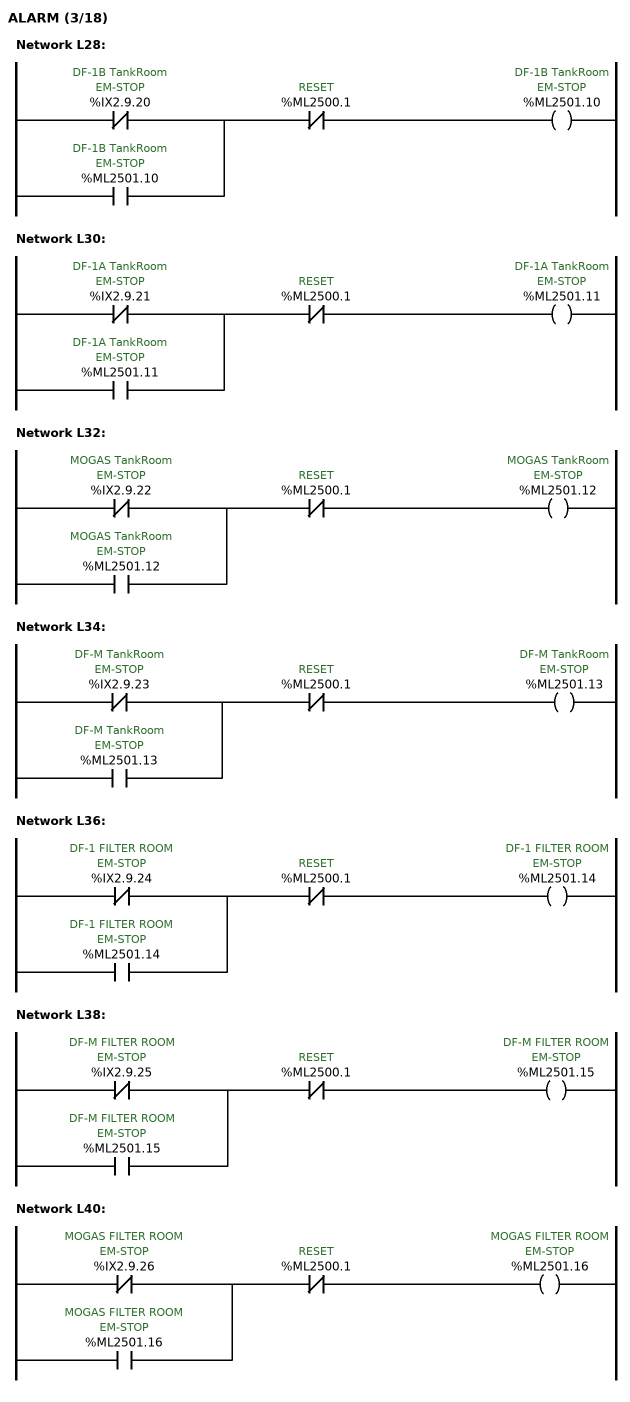
(* Rung L28 *)
%ML2501.10 := (NOT %IX2.9.20 OR %ML2501.10) AND NOT %ML2500.1;
(* Rung L30 *)
%ML2501.11 := (NOT %IX2.9.21 OR %ML2501.11) AND NOT %ML2500.1;
(* Rung L32 *)
%ML2501.12 := (NOT %IX2.9.22 OR %ML2501.12) AND NOT %ML2500.1;
(* Rung L34 *)
%ML2501.13 := (NOT %IX2.9.23 OR %ML2501.13) AND NOT %ML2500.1;
(* Rung L36 *)
%ML2501.14 := (NOT %IX2.9.24 OR %ML2501.14) AND NOT %ML2500.1;
(* Rung L38 *)
%ML2501.15 := (NOT %IX2.9.25 OR %ML2501.15) AND NOT %ML2500.1;
(* Rung L40 *)
%ML2501.16 := (NOT %IX2.9.26 OR %ML2501.16) AND NOT %ML2500.1;

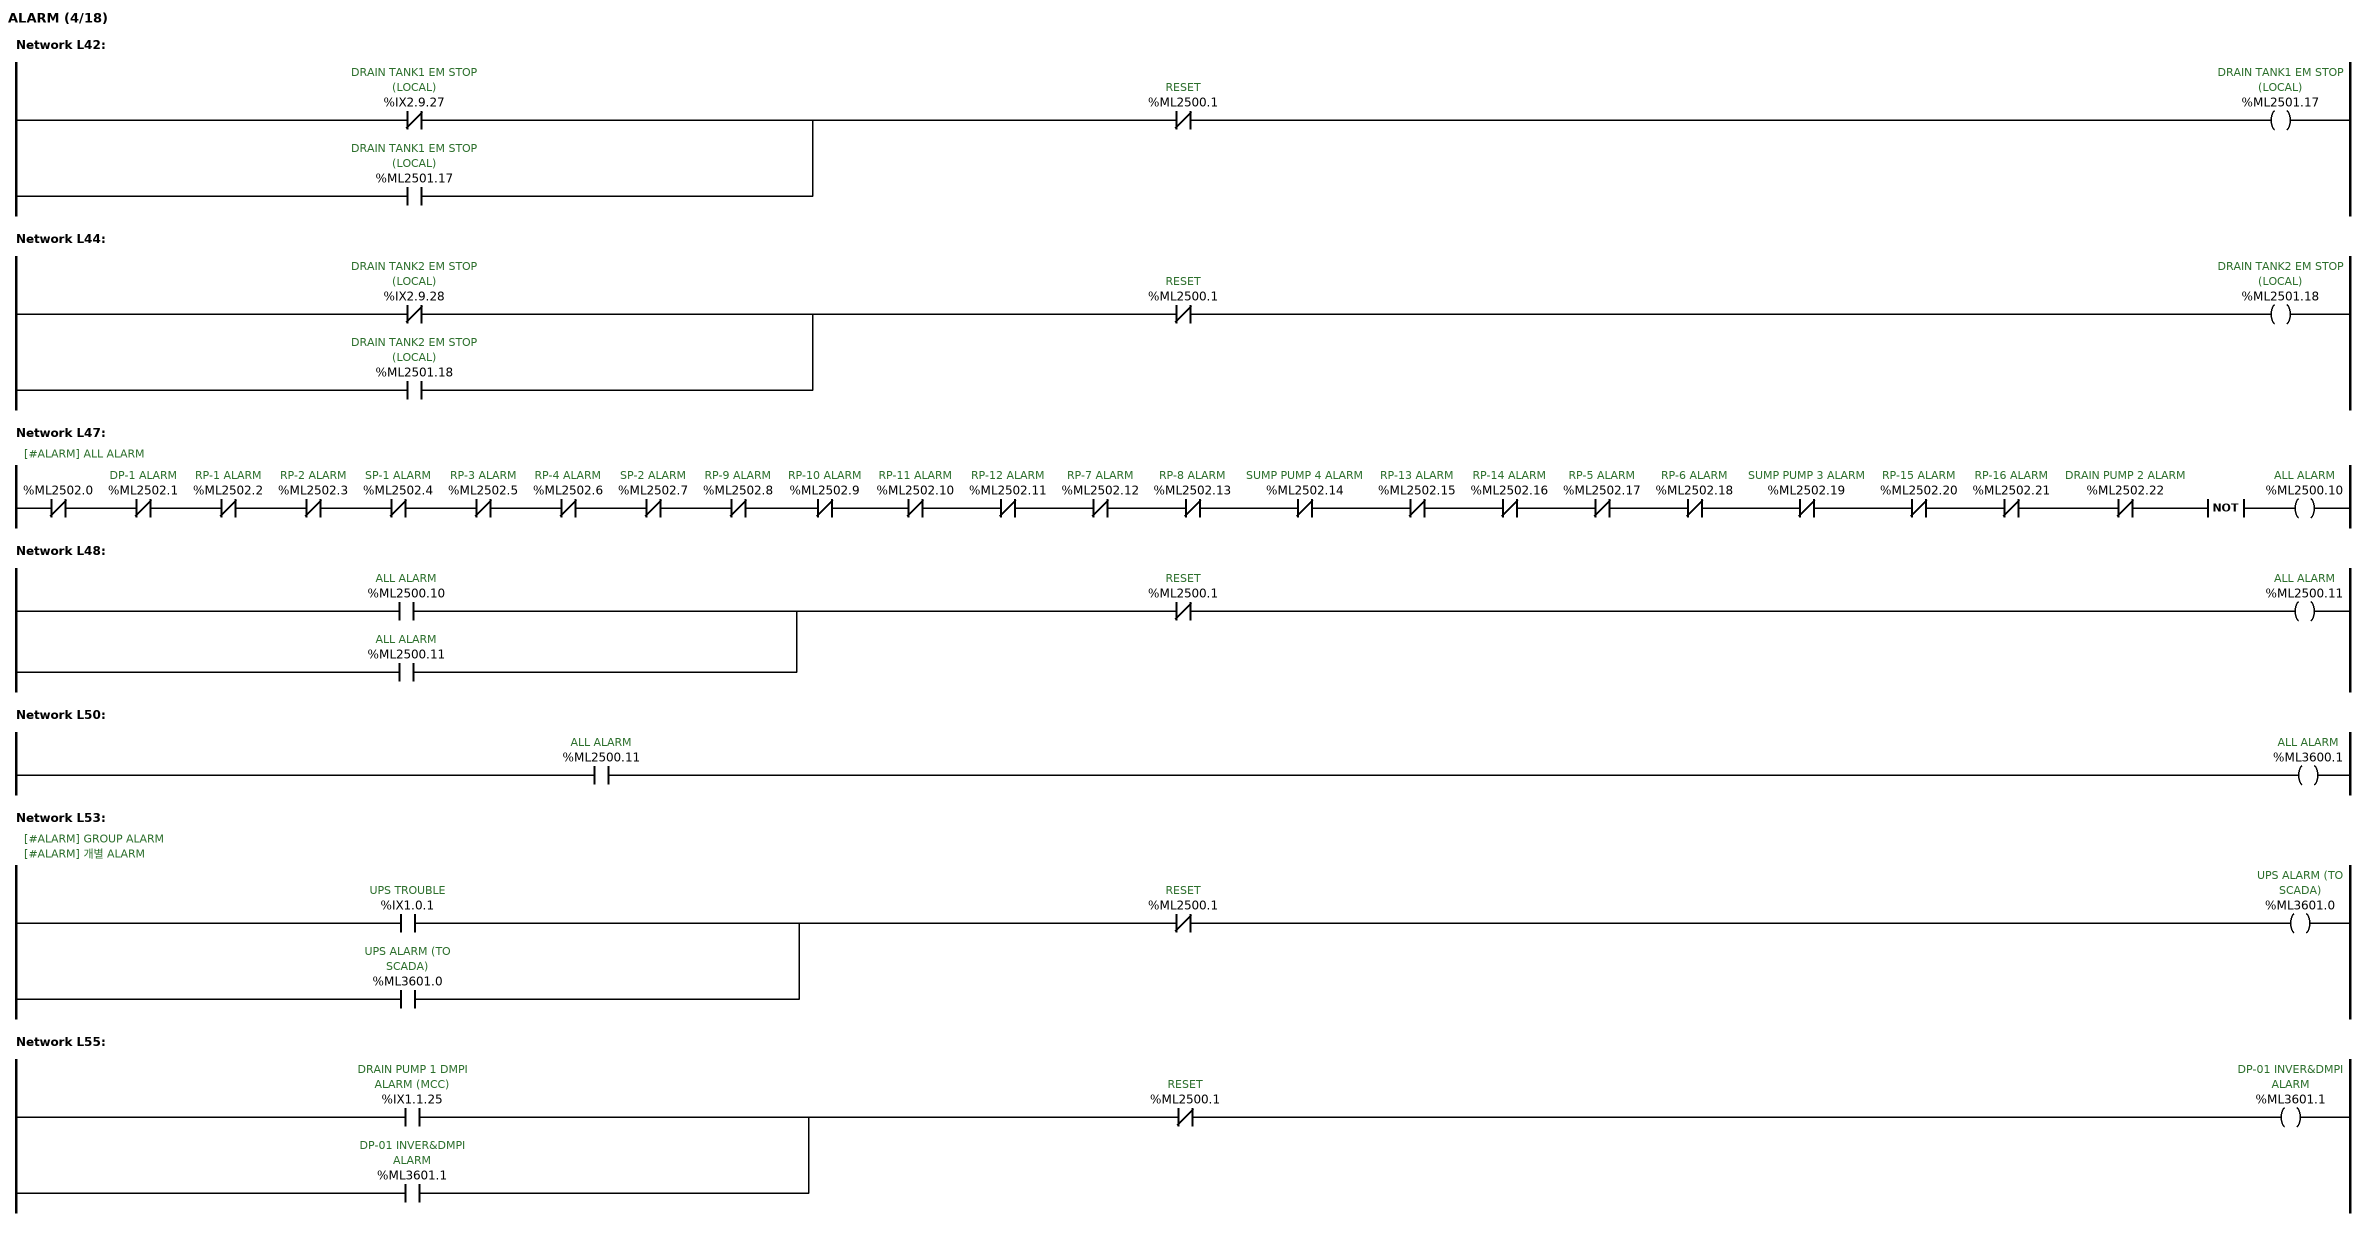
(* Rung L42 *)
%ML2501.17 := (NOT %IX2.9.27 OR %ML2501.17) AND NOT %ML2500.1;
(* Rung L44 *)
%ML2501.18 := (NOT %IX2.9.28 OR %ML2501.18) AND NOT %ML2500.1;
(* [#ALARM] ALL ALARM *)
(* Rung L47 *)
%ML2500.10 := NOT (NOT %ML2502.0 AND NOT %ML2502.1 AND NOT %ML2502.2 AND NOT %ML2502.3 AND NOT %ML2502.4 AND NOT %ML2502.5 AND NOT %ML2502.6 AND NOT %ML2502.7 AND NOT %ML2502.8 AND NOT %ML2502.9 AND NOT %ML2502.10 AND NOT %ML2502.11 AND NOT %ML2502.12 AND NOT %ML2502.13 AND NOT %ML2502.14 AND NOT %ML2502.15 AND NOT %ML2502.16 AND NOT %ML2502.17 AND NOT %ML2502.18 AND NOT %ML2502.19 AND NOT %ML2502.20 AND NOT %ML2502.21 AND NOT %ML2502.22);
(* Rung L48 *)
%ML2500.11 := (%ML2500.10 OR %ML2500.11) AND NOT %ML2500.1;
(* Rung L50 *)
%ML3600.1 := %ML2500.11;
(* [#ALARM] GROUP ALARM *)
(* [#ALARM] 개별 ALARM *)
(* Rung L53 *)
%ML3601.0 := (%IX1.0.1 OR %ML3601.0) AND NOT %ML2500.1;
(* Rung L55 *)
%ML3601.1 := (%IX1.1.25 OR %ML3601.1) AND NOT %ML2500.1;

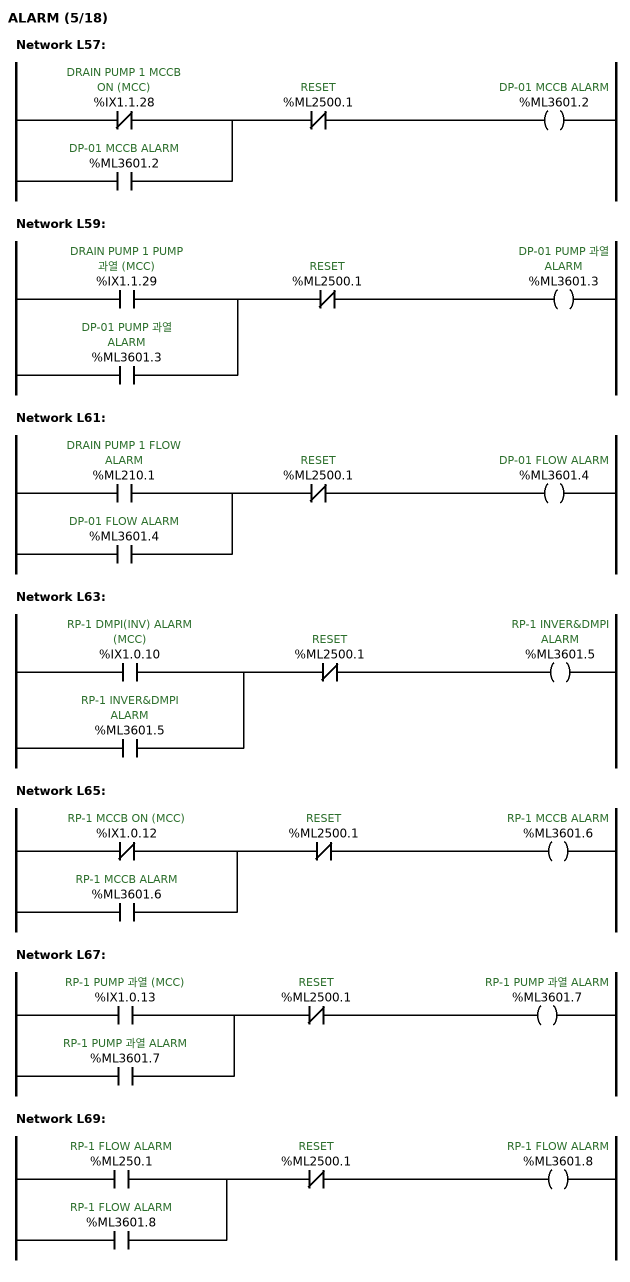
(* Rung L57 *)
%ML3601.2 := (NOT %IX1.1.28 OR %ML3601.2) AND NOT %ML2500.1;
(* Rung L59 *)
%ML3601.3 := (%IX1.1.29 OR %ML3601.3) AND NOT %ML2500.1;
(* Rung L61 *)
%ML3601.4 := (%ML210.1 OR %ML3601.4) AND NOT %ML2500.1;
(* Rung L63 *)
%ML3601.5 := (%IX1.0.10 OR %ML3601.5) AND NOT %ML2500.1;
(* Rung L65 *)
%ML3601.6 := (NOT %IX1.0.12 OR %ML3601.6) AND NOT %ML2500.1;
(* Rung L67 *)
%ML3601.7 := (%IX1.0.13 OR %ML3601.7) AND NOT %ML2500.1;
(* Rung L69 *)
%ML3601.8 := (%ML250.1 OR %ML3601.8) AND NOT %ML2500.1;

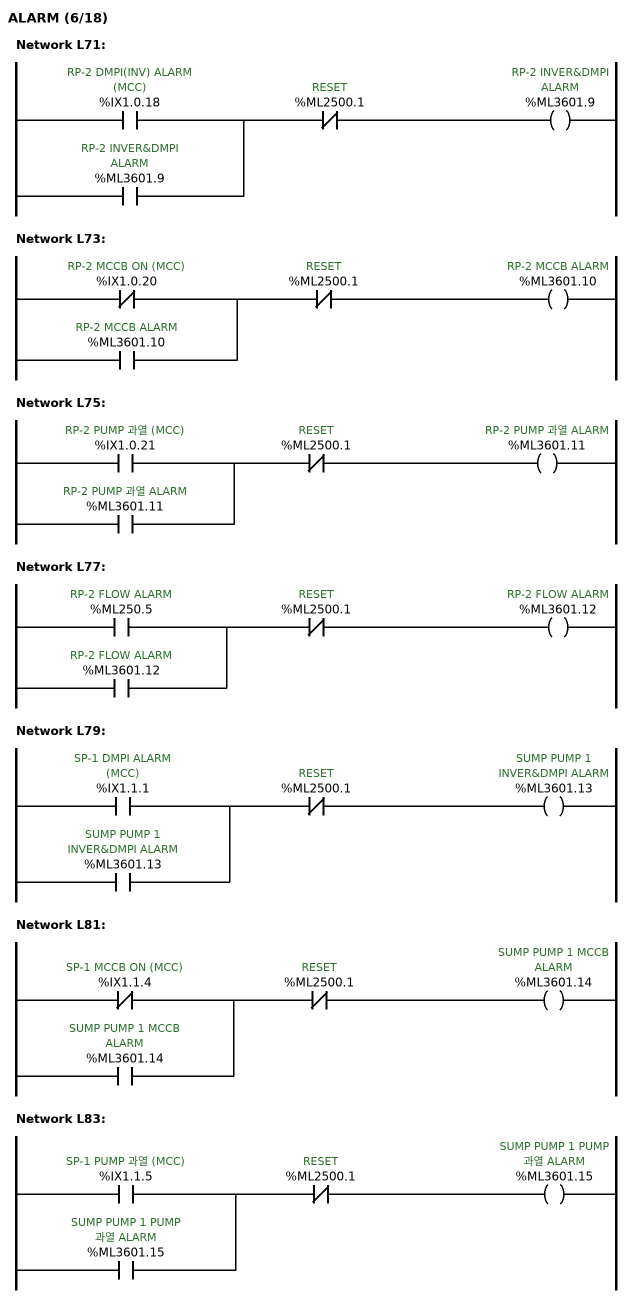
(* Rung L71 *)
%ML3601.9 := (%IX1.0.18 OR %ML3601.9) AND NOT %ML2500.1;
(* Rung L73 *)
%ML3601.10 := (NOT %IX1.0.20 OR %ML3601.10) AND NOT %ML2500.1;
(* Rung L75 *)
%ML3601.11 := (%IX1.0.21 OR %ML3601.11) AND NOT %ML2500.1;
(* Rung L77 *)
%ML3601.12 := (%ML250.5 OR %ML3601.12) AND NOT %ML2500.1;
(* Rung L79 *)
%ML3601.13 := (%IX1.1.1 OR %ML3601.13) AND NOT %ML2500.1;
(* Rung L81 *)
%ML3601.14 := (NOT %IX1.1.4 OR %ML3601.14) AND NOT %ML2500.1;
(* Rung L83 *)
%ML3601.15 := (%IX1.1.5 OR %ML3601.15) AND NOT %ML2500.1;

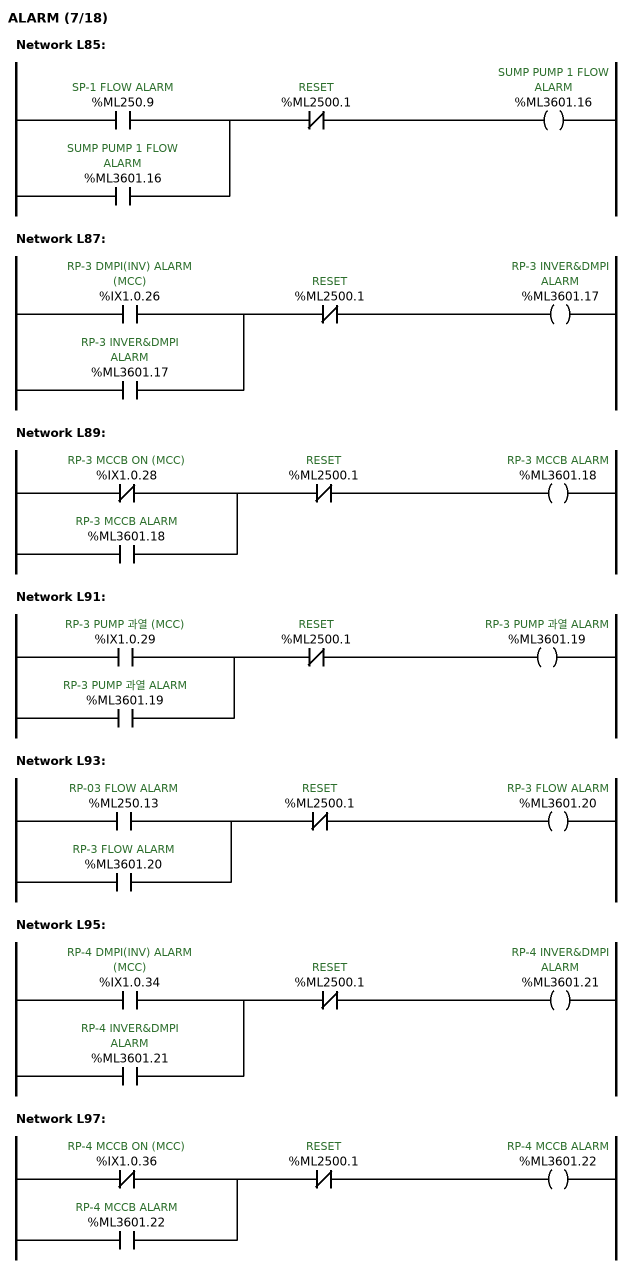
(* Rung L85 *)
%ML3601.16 := (%ML250.9 OR %ML3601.16) AND NOT %ML2500.1;
(* Rung L87 *)
%ML3601.17 := (%IX1.0.26 OR %ML3601.17) AND NOT %ML2500.1;
(* Rung L89 *)
%ML3601.18 := (NOT %IX1.0.28 OR %ML3601.18) AND NOT %ML2500.1;
(* Rung L91 *)
%ML3601.19 := (%IX1.0.29 OR %ML3601.19) AND NOT %ML2500.1;
(* Rung L93 *)
%ML3601.20 := (%ML250.13 OR %ML3601.20) AND NOT %ML2500.1;
(* Rung L95 *)
%ML3601.21 := (%IX1.0.34 OR %ML3601.21) AND NOT %ML2500.1;
(* Rung L97 *)
%ML3601.22 := (NOT %IX1.0.36 OR %ML3601.22) AND NOT %ML2500.1;

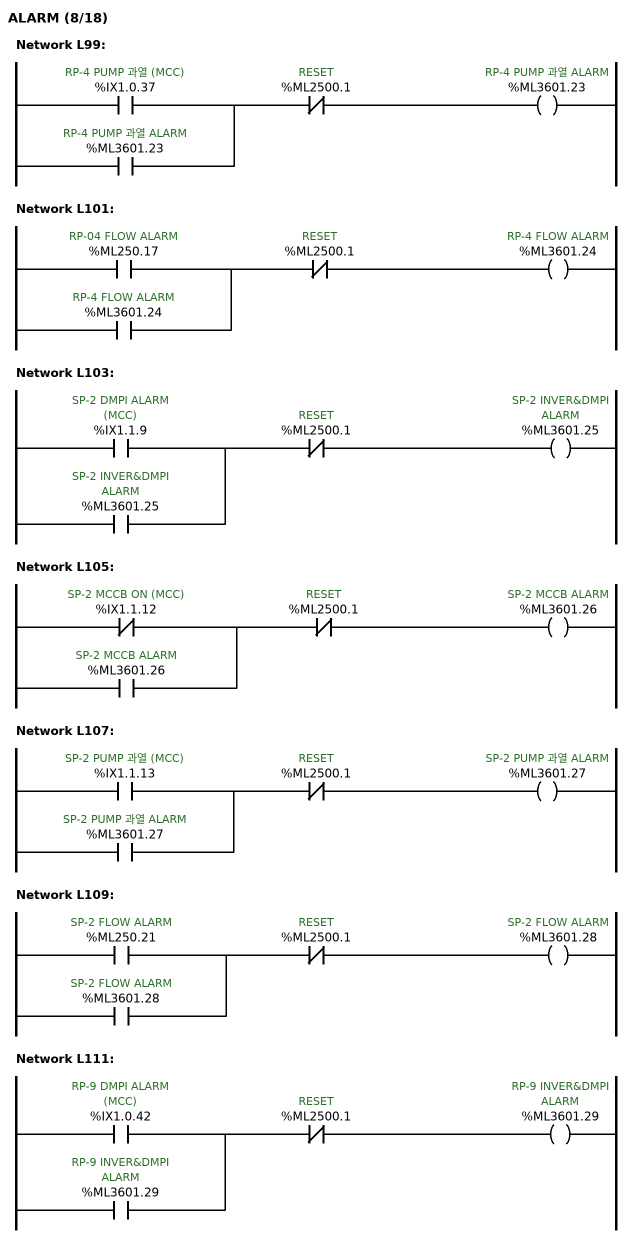
(* Rung L99 *)
%ML3601.23 := (%IX1.0.37 OR %ML3601.23) AND NOT %ML2500.1;
(* Rung L101 *)
%ML3601.24 := (%ML250.17 OR %ML3601.24) AND NOT %ML2500.1;
(* Rung L103 *)
%ML3601.25 := (%IX1.1.9 OR %ML3601.25) AND NOT %ML2500.1;
(* Rung L105 *)
%ML3601.26 := (NOT %IX1.1.12 OR %ML3601.26) AND NOT %ML2500.1;
(* Rung L107 *)
%ML3601.27 := (%IX1.1.13 OR %ML3601.27) AND NOT %ML2500.1;
(* Rung L109 *)
%ML3601.28 := (%ML250.21 OR %ML3601.28) AND NOT %ML2500.1;
(* Rung L111 *)
%ML3601.29 := (%IX1.0.42 OR %ML3601.29) AND NOT %ML2500.1;

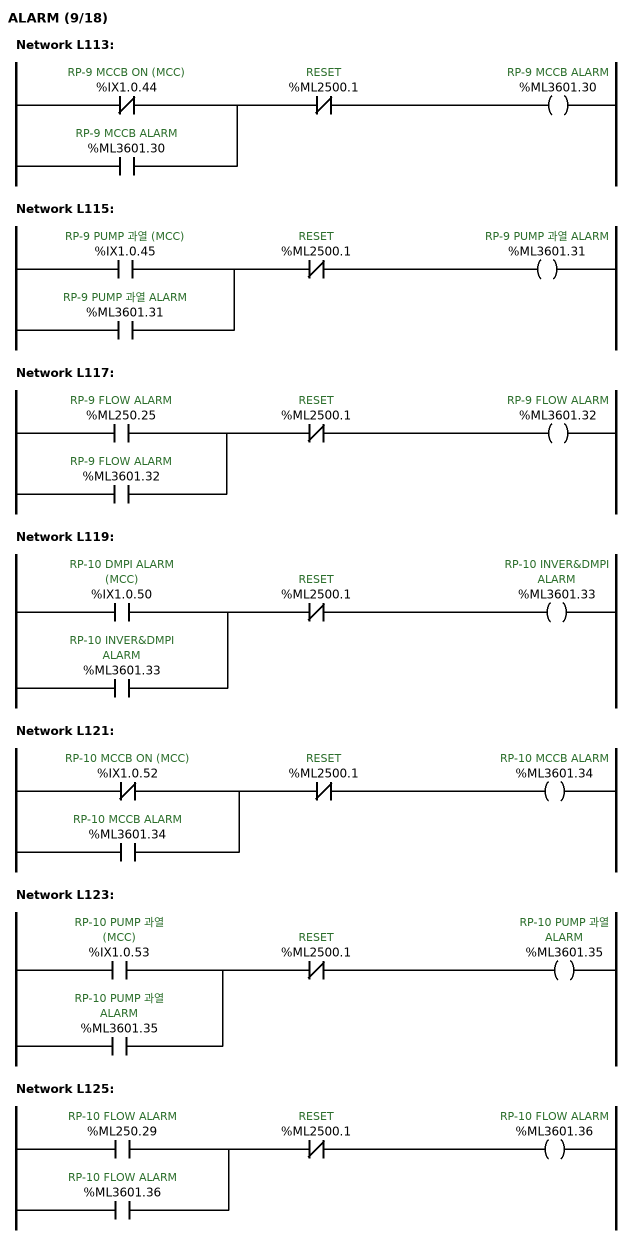
(* Rung L113 *)
%ML3601.30 := (NOT %IX1.0.44 OR %ML3601.30) AND NOT %ML2500.1;
(* Rung L115 *)
%ML3601.31 := (%IX1.0.45 OR %ML3601.31) AND NOT %ML2500.1;
(* Rung L117 *)
%ML3601.32 := (%ML250.25 OR %ML3601.32) AND NOT %ML2500.1;
(* Rung L119 *)
%ML3601.33 := (%IX1.0.50 OR %ML3601.33) AND NOT %ML2500.1;
(* Rung L121 *)
%ML3601.34 := (NOT %IX1.0.52 OR %ML3601.34) AND NOT %ML2500.1;
(* Rung L123 *)
%ML3601.35 := (%IX1.0.53 OR %ML3601.35) AND NOT %ML2500.1;
(* Rung L125 *)
%ML3601.36 := (%ML250.29 OR %ML3601.36) AND NOT %ML2500.1;

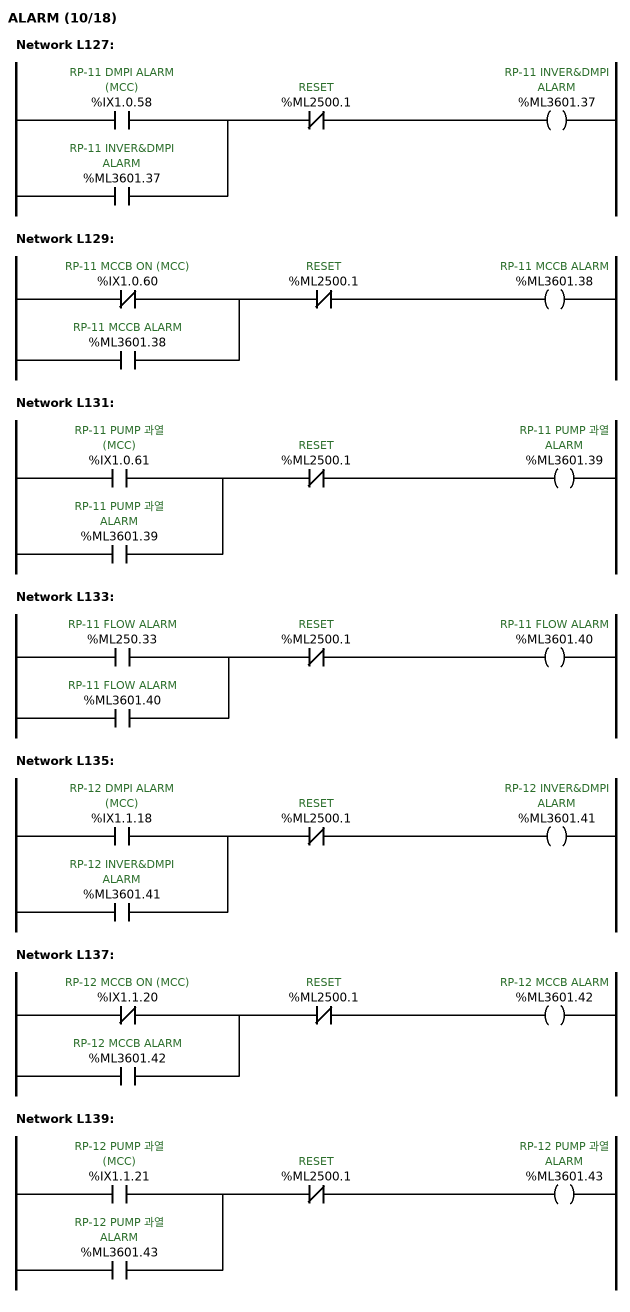
(* Rung L127 *)
%ML3601.37 := (%IX1.0.58 OR %ML3601.37) AND NOT %ML2500.1;
(* Rung L129 *)
%ML3601.38 := (NOT %IX1.0.60 OR %ML3601.38) AND NOT %ML2500.1;
(* Rung L131 *)
%ML3601.39 := (%IX1.0.61 OR %ML3601.39) AND NOT %ML2500.1;
(* Rung L133 *)
%ML3601.40 := (%ML250.33 OR %ML3601.40) AND NOT %ML2500.1;
(* Rung L135 *)
%ML3601.41 := (%IX1.1.18 OR %ML3601.41) AND NOT %ML2500.1;
(* Rung L137 *)
%ML3601.42 := (NOT %IX1.1.20 OR %ML3601.42) AND NOT %ML2500.1;
(* Rung L139 *)
%ML3601.43 := (%IX1.1.21 OR %ML3601.43) AND NOT %ML2500.1;

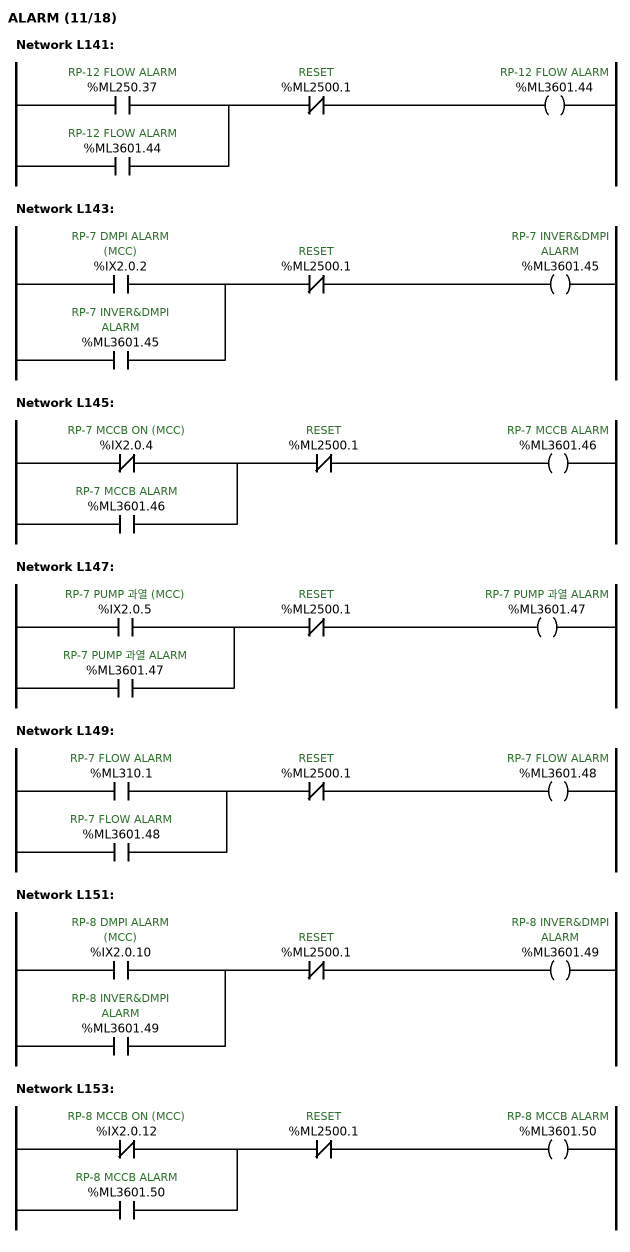
(* Rung L141 *)
%ML3601.44 := (%ML250.37 OR %ML3601.44) AND NOT %ML2500.1;
(* Rung L143 *)
%ML3601.45 := (%IX2.0.2 OR %ML3601.45) AND NOT %ML2500.1;
(* Rung L145 *)
%ML3601.46 := (NOT %IX2.0.4 OR %ML3601.46) AND NOT %ML2500.1;
(* Rung L147 *)
%ML3601.47 := (%IX2.0.5 OR %ML3601.47) AND NOT %ML2500.1;
(* Rung L149 *)
%ML3601.48 := (%ML310.1 OR %ML3601.48) AND NOT %ML2500.1;
(* Rung L151 *)
%ML3601.49 := (%IX2.0.10 OR %ML3601.49) AND NOT %ML2500.1;
(* Rung L153 *)
%ML3601.50 := (NOT %IX2.0.12 OR %ML3601.50) AND NOT %ML2500.1;

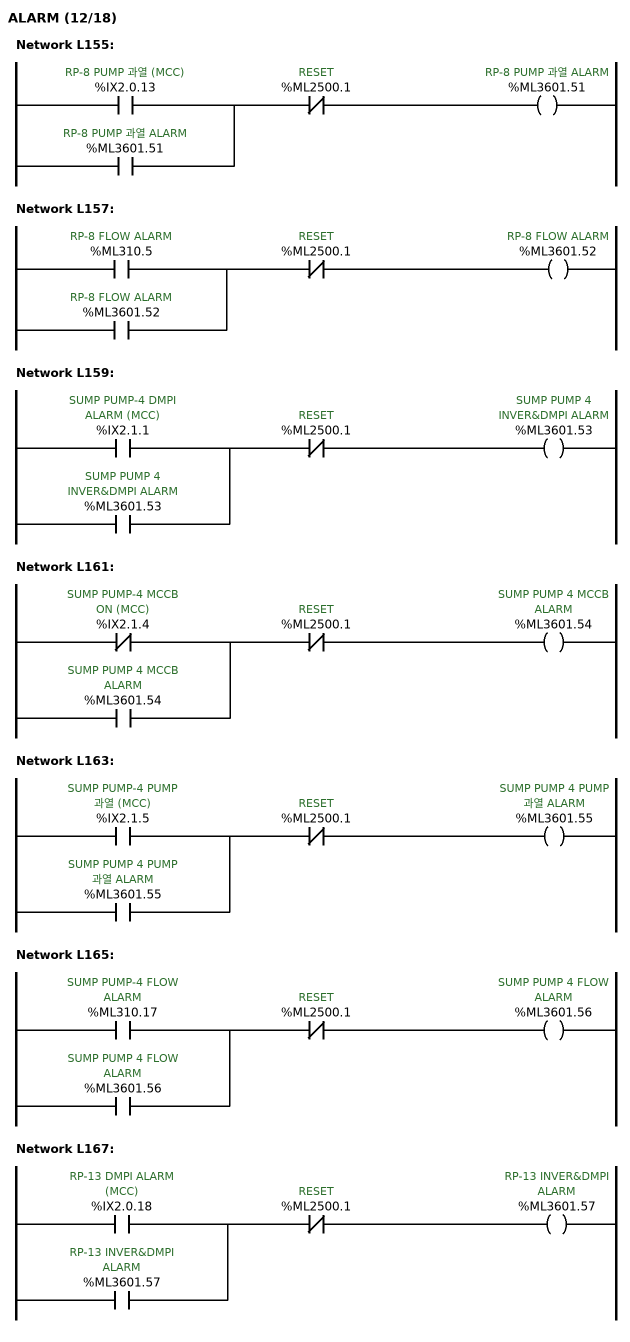
(* Rung L155 *)
%ML3601.51 := (%IX2.0.13 OR %ML3601.51) AND NOT %ML2500.1;
(* Rung L157 *)
%ML3601.52 := (%ML310.5 OR %ML3601.52) AND NOT %ML2500.1;
(* Rung L159 *)
%ML3601.53 := (%IX2.1.1 OR %ML3601.53) AND NOT %ML2500.1;
(* Rung L161 *)
%ML3601.54 := (NOT %IX2.1.4 OR %ML3601.54) AND NOT %ML2500.1;
(* Rung L163 *)
%ML3601.55 := (%IX2.1.5 OR %ML3601.55) AND NOT %ML2500.1;
(* Rung L165 *)
%ML3601.56 := (%ML310.17 OR %ML3601.56) AND NOT %ML2500.1;
(* Rung L167 *)
%ML3601.57 := (%IX2.0.18 OR %ML3601.57) AND NOT %ML2500.1;

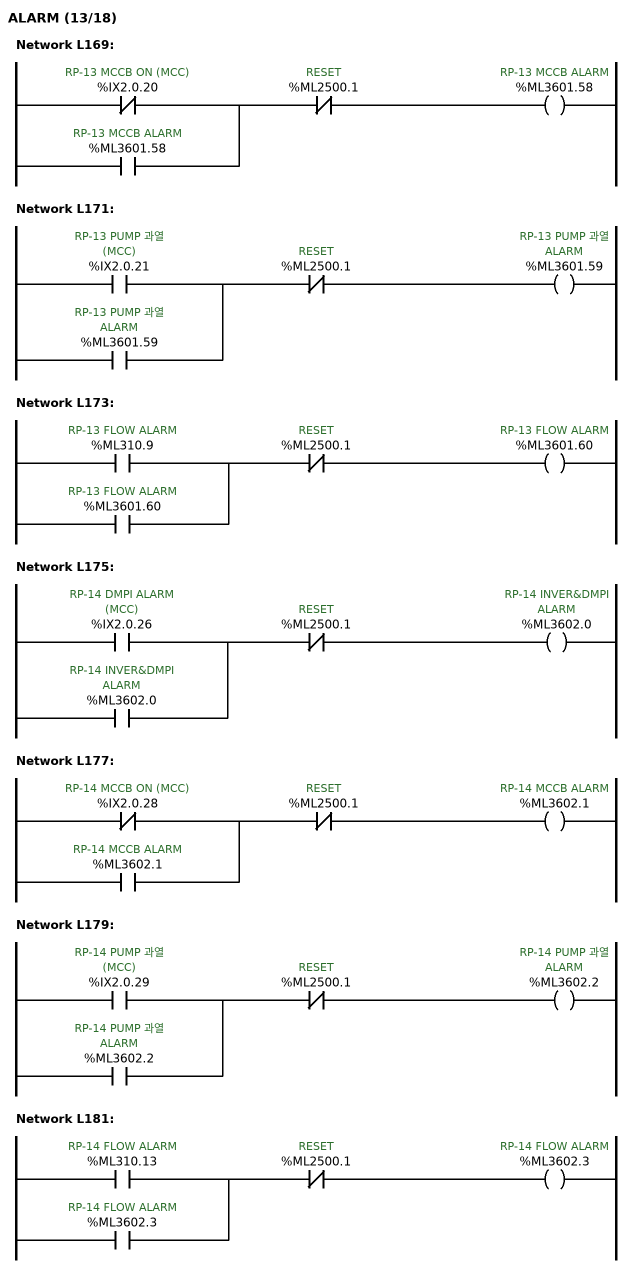
(* Rung L169 *)
%ML3601.58 := (NOT %IX2.0.20 OR %ML3601.58) AND NOT %ML2500.1;
(* Rung L171 *)
%ML3601.59 := (%IX2.0.21 OR %ML3601.59) AND NOT %ML2500.1;
(* Rung L173 *)
%ML3601.60 := (%ML310.9 OR %ML3601.60) AND NOT %ML2500.1;
(* Rung L175 *)
%ML3602.0 := (%IX2.0.26 OR %ML3602.0) AND NOT %ML2500.1;
(* Rung L177 *)
%ML3602.1 := (NOT %IX2.0.28 OR %ML3602.1) AND NOT %ML2500.1;
(* Rung L179 *)
%ML3602.2 := (%IX2.0.29 OR %ML3602.2) AND NOT %ML2500.1;
(* Rung L181 *)
%ML3602.3 := (%ML310.13 OR %ML3602.3) AND NOT %ML2500.1;

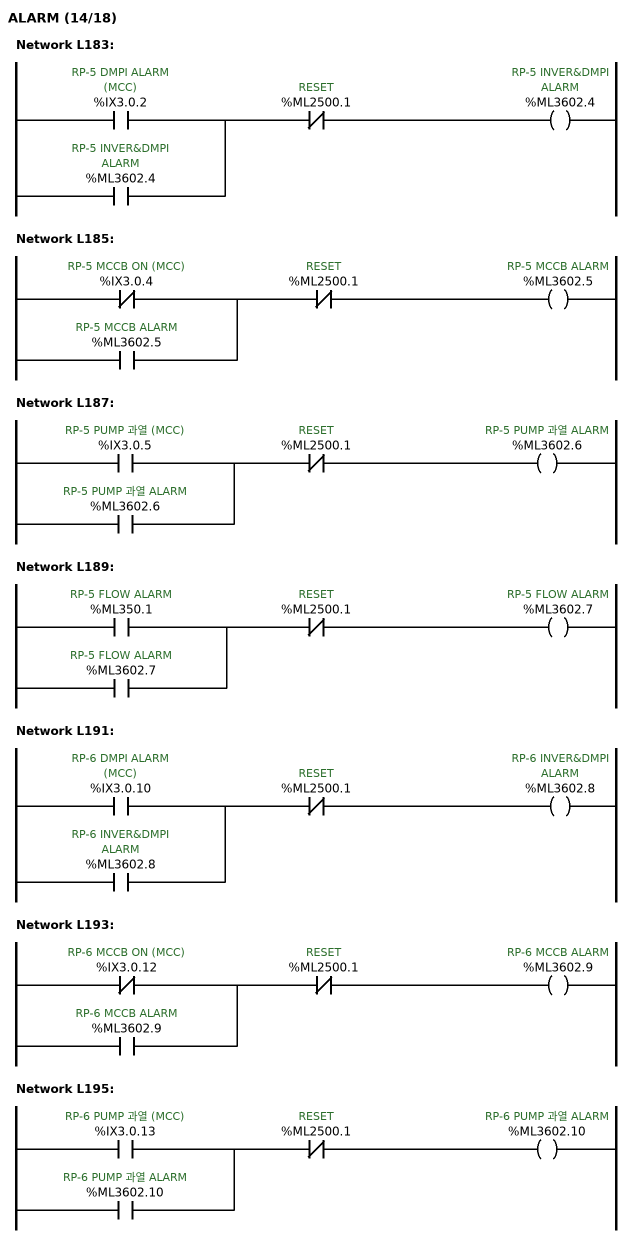
(* Rung L183 *)
%ML3602.4 := (%IX3.0.2 OR %ML3602.4) AND NOT %ML2500.1;
(* Rung L185 *)
%ML3602.5 := (NOT %IX3.0.4 OR %ML3602.5) AND NOT %ML2500.1;
(* Rung L187 *)
%ML3602.6 := (%IX3.0.5 OR %ML3602.6) AND NOT %ML2500.1;
(* Rung L189 *)
%ML3602.7 := (%ML350.1 OR %ML3602.7) AND NOT %ML2500.1;
(* Rung L191 *)
%ML3602.8 := (%IX3.0.10 OR %ML3602.8) AND NOT %ML2500.1;
(* Rung L193 *)
%ML3602.9 := (NOT %IX3.0.12 OR %ML3602.9) AND NOT %ML2500.1;
(* Rung L195 *)
%ML3602.10 := (%IX3.0.13 OR %ML3602.10) AND NOT %ML2500.1;

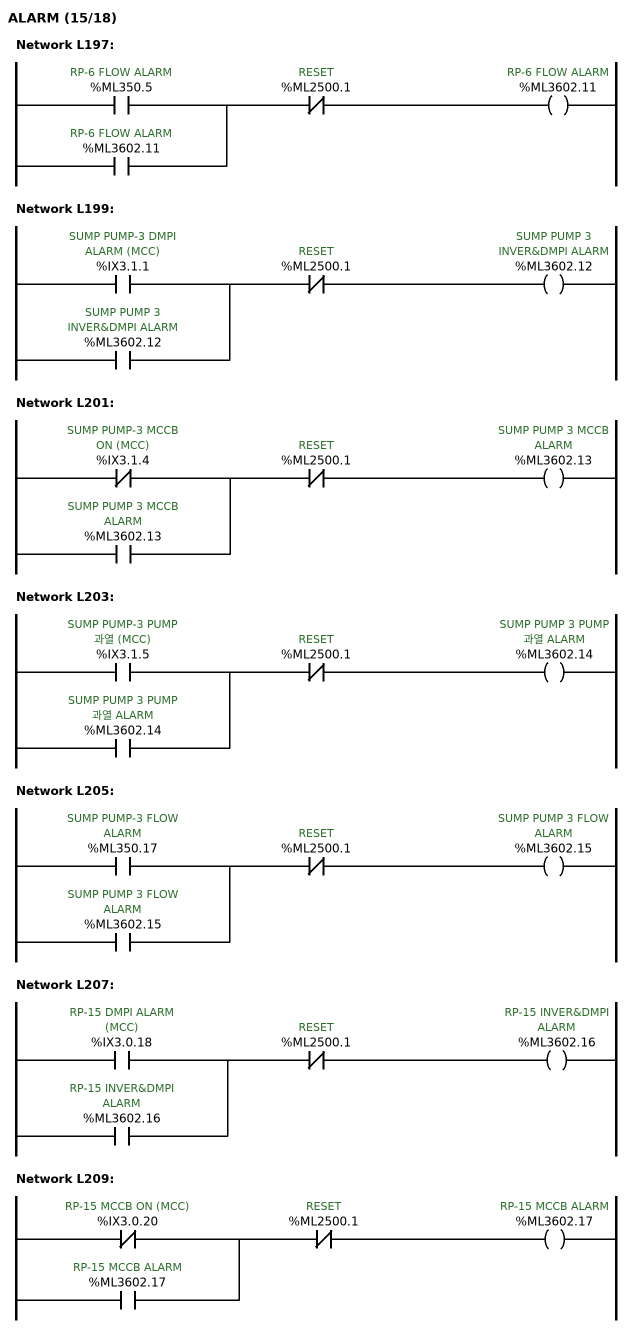
(* Rung L197 *)
%ML3602.11 := (%ML350.5 OR %ML3602.11) AND NOT %ML2500.1;
(* Rung L199 *)
%ML3602.12 := (%IX3.1.1 OR %ML3602.12) AND NOT %ML2500.1;
(* Rung L201 *)
%ML3602.13 := (NOT %IX3.1.4 OR %ML3602.13) AND NOT %ML2500.1;
(* Rung L203 *)
%ML3602.14 := (%IX3.1.5 OR %ML3602.14) AND NOT %ML2500.1;
(* Rung L205 *)
%ML3602.15 := (%ML350.17 OR %ML3602.15) AND NOT %ML2500.1;
(* Rung L207 *)
%ML3602.16 := (%IX3.0.18 OR %ML3602.16) AND NOT %ML2500.1;
(* Rung L209 *)
%ML3602.17 := (NOT %IX3.0.20 OR %ML3602.17) AND NOT %ML2500.1;

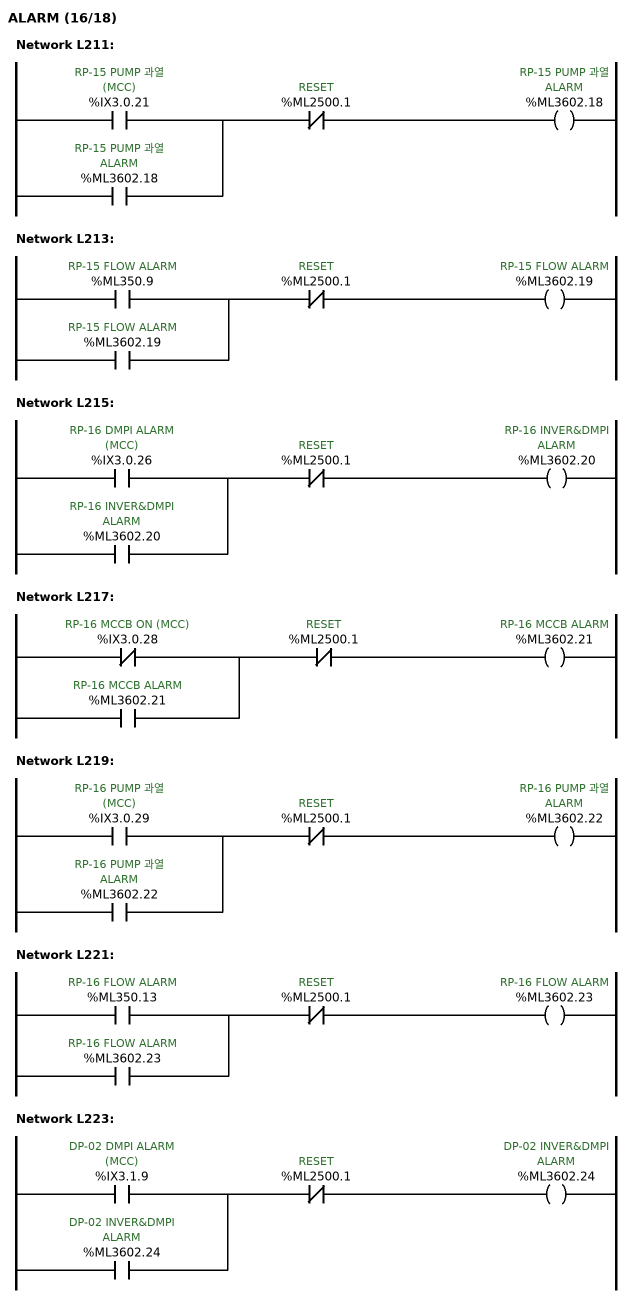
(* Rung L211 *)
%ML3602.18 := (%IX3.0.21 OR %ML3602.18) AND NOT %ML2500.1;
(* Rung L213 *)
%ML3602.19 := (%ML350.9 OR %ML3602.19) AND NOT %ML2500.1;
(* Rung L215 *)
%ML3602.20 := (%IX3.0.26 OR %ML3602.20) AND NOT %ML2500.1;
(* Rung L217 *)
%ML3602.21 := (NOT %IX3.0.28 OR %ML3602.21) AND NOT %ML2500.1;
(* Rung L219 *)
%ML3602.22 := (%IX3.0.29 OR %ML3602.22) AND NOT %ML2500.1;
(* Rung L221 *)
%ML3602.23 := (%ML350.13 OR %ML3602.23) AND NOT %ML2500.1;
(* Rung L223 *)
%ML3602.24 := (%IX3.1.9 OR %ML3602.24) AND NOT %ML2500.1;

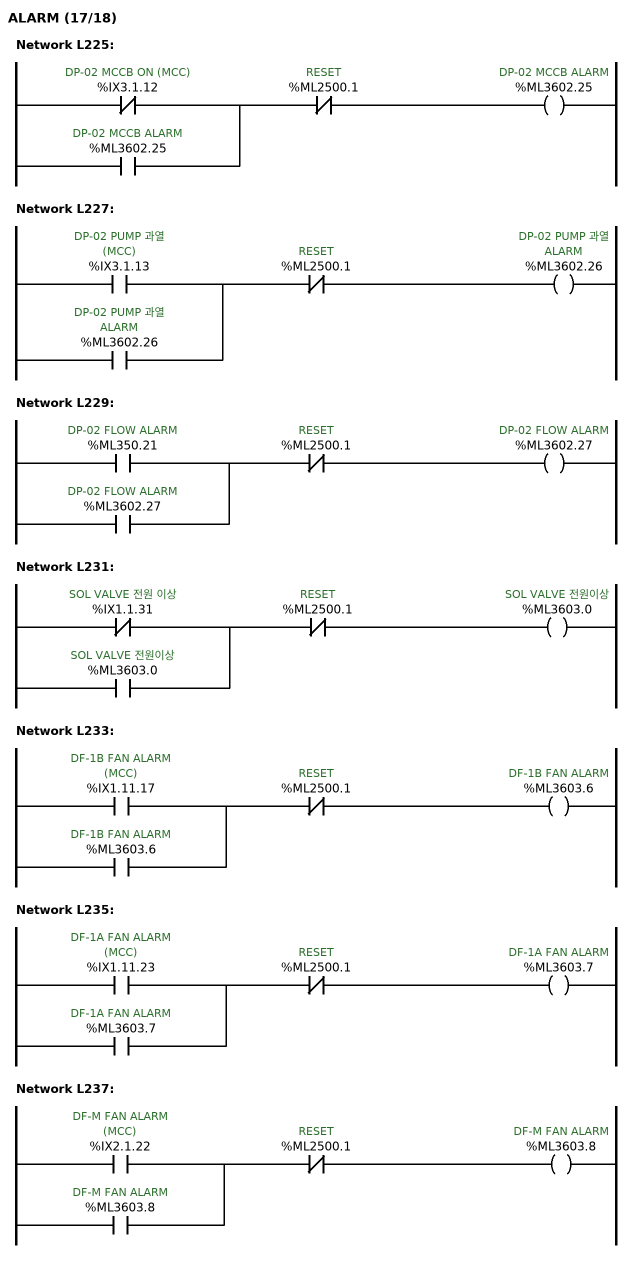
(* Rung L225 *)
%ML3602.25 := (NOT %IX3.1.12 OR %ML3602.25) AND NOT %ML2500.1;
(* Rung L227 *)
%ML3602.26 := (%IX3.1.13 OR %ML3602.26) AND NOT %ML2500.1;
(* Rung L229 *)
%ML3602.27 := (%ML350.21 OR %ML3602.27) AND NOT %ML2500.1;
(* Rung L231 *)
%ML3603.0 := (NOT %IX1.1.31 OR %ML3603.0) AND NOT %ML2500.1;
(* Rung L233 *)
%ML3603.6 := (%IX1.11.17 OR %ML3603.6) AND NOT %ML2500.1;
(* Rung L235 *)
%ML3603.7 := (%IX1.11.23 OR %ML3603.7) AND NOT %ML2500.1;
(* Rung L237 *)
%ML3603.8 := (%IX2.1.22 OR %ML3603.8) AND NOT %ML2500.1;

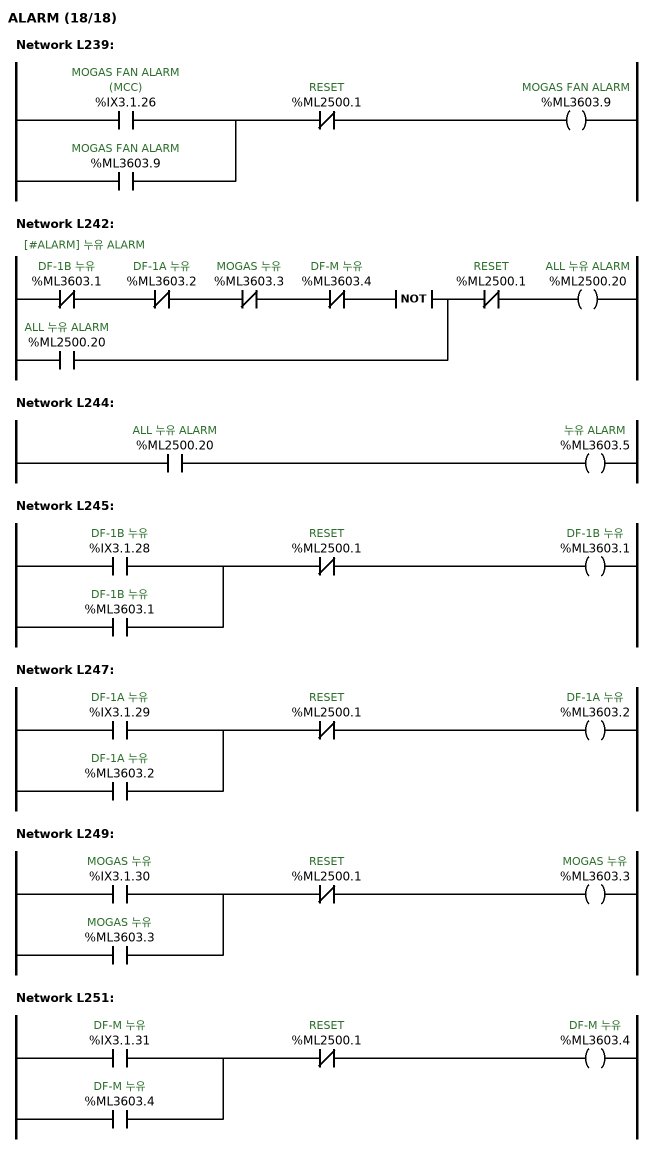
(* Rung L239 *)
%ML3603.9 := (%IX3.1.26 OR %ML3603.9) AND NOT %ML2500.1;
(* [#ALARM] 누유 ALARM *)
(* Rung L242 *)
%ML2500.20 := (NOT (NOT %ML3603.1 AND NOT %ML3603.2 AND NOT %ML3603.3 AND NOT %ML3603.4) OR %ML2500.20) AND NOT %ML2500.1;
(* Rung L244 *)
%ML3603.5 := %ML2500.20;
(* Rung L245 *)
%ML3603.1 := (%IX3.1.28 OR %ML3603.1) AND NOT %ML2500.1;
(* Rung L247 *)
%ML3603.2 := (%IX3.1.29 OR %ML3603.2) AND NOT %ML2500.1;
(* Rung L249 *)
%ML3603.3 := (%IX3.1.30 OR %ML3603.3) AND NOT %ML2500.1;
(* Rung L251 *)
%ML3603.4 := (%IX3.1.31 OR %ML3603.4) AND NOT %ML2500.1;
END_PROGRAM